// Mitsubishi GX Works2 project: ex01   PLC: Q02/Q02H

PROGRAM MAIN
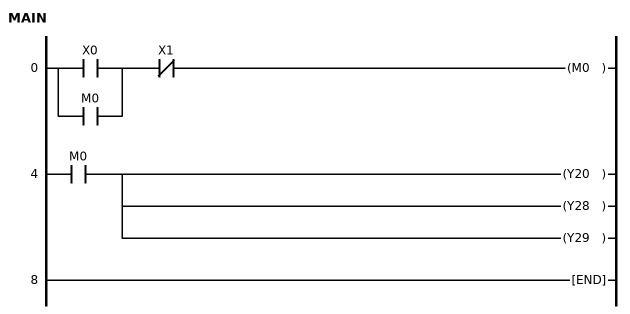
0     LD      X0
      OR      M0
      ANI     X1
      OUT     M0
4     LD      M0
      OUT     Y20
      OUT     Y28
      OUT     Y29
8     END
END_PROGRAM
